(* Logix 5000 project; controller Amvex_Thorpe_Flowmeter vendor 1 type 14 code 106 rev 33.13; software revision 33.01 *)

TASK MainTask (continuous, watchdog 500 ms) : MainProgram
TASK MCP_TESTING_STATION (periodic, rate 10 ms, priority 10, watchdog 500 ms) : MCP_Main
TASK RCP1_FITTING_STATION (periodic, rate 10 ms, priority 10, watchdog 500 ms) : RPC1_Main

MODULES
   Local : vendor 1 type 14 code 106 (Compact 0, rev 33.13)
      RCP1_Valve_Stack : EX260-SEN1 (Ethernet 192.168.30.96, rev 1.1, Output RPI 10 ms)
      MCP_VALVE_STACK : EX260-SEN1 (Ethernet 192.168.30.110, rev 1.1, Output RPI 10 ms)
           MCP_VALVE_STACK:O.OutputArea[0].10   // VB1.O.Sol_A.5
           MCP_VALVE_STACK:O.OutputArea[0].0   // VB1.O.Sol_A.0
           MCP_VALVE_STACK:O.OutputArea[0].1   // VB1.O.Sol_B.0
           MCP_VALVE_STACK:O.OutputArea[0].2   // VB1.O.Sol_A.1
           MCP_VALVE_STACK:O.OutputArea[0].3   // VB1.O.Sol_B.1
           MCP_VALVE_STACK:O.OutputArea[0].4   // VB1.O.Sol_A.2
           MCP_VALVE_STACK:O.OutputArea[0].5   // VB1.O.Sol_B.2
           MCP_VALVE_STACK:O.OutputArea[0].6   // VB1.O.Sol_A.3
           MCP_VALVE_STACK:O.OutputArea[0].7   // VB1.O.Sol_B.3
           MCP_VALVE_STACK:O.OutputArea[0].8   // VB1.O.Sol_A.4
           MCP_VALVE_STACK:O.OutputArea[0].9   // VB1.O.Sol_B.4
           MCP_VALVE_STACK:O.OutputArea[1].0   // VB1.O.Sol_A.8
           MCP_VALVE_STACK:O.OutputArea[1].1   // VB1.O.Sol_B.8
           MCP_VALVE_STACK:O.OutputArea[0].11   // VB1.O.Sol_B.5
           MCP_VALVE_STACK:O.OutputArea[0].12   // VB1.O.Sol_A.6
           MCP_VALVE_STACK:O.OutputArea[0].13   // VB1.O.Sol_B.6
           MCP_VALVE_STACK:O.OutputArea[0].14   // VB1.O.Sol_A.7
           MCP_VALVE_STACK:O.OutputArea[0].15   // VB1.O.Sol_B.7
           MCP_VALVE_STACK:O.OutputArea[1].2   // VB1.O.Sol_A.9
           MCP_VALVE_STACK:O.OutputArea[1].3   // VB1.O.Sol_B.9
      MCP_00 : 1334920000 (Ethernet 192.168.30.101, rev 1.6, StandardDataDriven RPI 10 ms)   // MCP - RR00 - ADAPTER MODULE 00
      Knob_Turner : SV2-CM-ENETIP (Ethernet 192.168.30.115, rev 1.1, StandardDataDriven RPI 10 ms)
           Knob_Turner:I.Data[4]   // Path Status
           Knob_Turner:I.Data[3].4   // Target position reached
           Knob_Turner:I.Data[3].5   // Torque limit active
           Knob_Turner:I.Data[0]   // Torque Feedback
           Knob_Turner:I.Data[1]   // Speed Feedback
           Knob_Turner:I.Data[2]   // Position Error
           Knob_Turner:I.Data[3].2   // Zero Speed
           Knob_Turner:I.Data[3].1   // Servo ON
           Knob_Turner:I.Data[3].0   // Ready
           Knob_Turner:I.Data[3].3   // Target speed reached
           Knob_Turner:I.Data[3].9   // Early overload warnining
           Knob_Turner:I.Data[3]   // General Outputs
           Knob_Turner:I.Data[3].6   // Alarm
           Knob_Turner:I.Data[3].8   // Home Complete
           Knob_Turner:I.Data[3].10   // Warning
           Knob_Turner:I.Data[3].7   // Brake
           Knob_Turner:O.Data[2].1   // Pulse clear
           Knob_Turner:O.Data[3]   // Path target
           Knob_Turner:O.Data[7]   // Path 1 data
           Knob_Turner:O.Data[8]   // Path 2 data
           Knob_Turner:O.Data[2].4   // Alarm reset
           Knob_Turner:O.Data[9]   // Path 3 data
           Knob_Turner:O.Data[2]   // DI control
           Knob_Turner:O.Data[2].7   // Motor Stop
           Knob_Turner:O.Data[2].0   // Servo on
           Knob_Turner:O.Data[2].2   // Torque 1
           Knob_Turner:O.Data[2].3   // Torque 2
           Knob_Turner:O.Data[4]   // Path trigger
           Knob_Turner:O.Data[1]   // DI control switch
           Knob_Turner:O.Data[2].5   // Rev inhibit limit
           Knob_Turner:O.Data[2].6   // Forw inhitibit limit
           Knob_Turner:O.Data[5]   // Speed 1
           Knob_Turner:O.Data[11]   // Torque limit 1
           Knob_Turner:O.Data[12]   // Torque limit 2
           Knob_Turner:O.Data[0]   // Aux functions
           Knob_Turner:O.Data[10]   // Path 4 data
           Knob_Turner:O.Data[6]   // Speed 2
      MCP_SAFETY_CTL : XS26 SC26 SC10 (Ethernet 192.168.30.104, rev 2.1, StandardDataDriven RPI 100 ms, StandardDataDriven RPI 100 ms)
      RCP1_SAFETY_CTL : XS26 SC26 SC10 (Ethernet 192.168.30.93, rev 2.1, StandardDataDriven RPI 100 ms, StandardDataDriven RPI 100 ms)
      IV3 : IV3 Series (Ethernet 192.168.30.106, rev 1.1, StandardDataDriven RPI 25 ms)
           IV3:I.Data[134]   // Tool 10 number of pitches, color average V (brightness), brightness average
           IV3:I.Data[0].1   // Master image regestration response
           IV3:I.Data[144]   // Tool 11 number of pitches, color average V (brightness), brightness average
           IV3:I.Data[154]   // Tool 12 number of pitches, color average V (brightness), brightness average
           IV3:I.Data[36]   // Tool 1 matching rate
           IV3:I.Data[46]   // Tool 2 matching rate
           IV3:I.Data[164]   // Tool 13 number of pitches, color average V (brightness), brightness average
           IV3:I.Data[174]   // Tool 14 number of pitches, color average V (brightness), brightness average
           IV3:I.Data[44]   // Tool 1 number of pitches, color average V (brightness), brightness average
           IV3:I.Data[56]   // Tool 3 matching rate
           IV3:I.Data[42]   // Tool 1 pitch present value MAX, color average H (hue)
           IV3:I.Data[52]   // Tool 2 pitch present value MAX, color average H (hue)
           IV3:I.Data[104]   // Tool 7 number of pitches, color average V (brightness), brightness average
           IV3:I.Data[0].15   // Setting value change failed
           IV3:I.Data[1].12   // Insufficient free space on SD card
           IV3:I.Data[2].0   // Overall judgment OK
           IV3:I.Data[129]   // Tool 10 lower threshold
           IV3:I.Data[130]   // Tool 10 upper threshold
           IV3:I.Data[12]   // Processing time MAX
           IV3:I.Data[0].3   // Warning clear response
           IV3:I.Data[100]   // Tool 7 upper threshold
           IV3:I.Data[26]   // Position adjustment tool matching rate
           IV3:I.Data[20]   // Number of NGs (standard mode/sorting mode)
           IV3:I.Data[21]   // Number of NGs (standard mode/sorting mode)
           IV3:I.Data[15]   // Reserved
           IV3:I.Data[24]   // Reserved
           IV3:I.Data[25]   // Reserved
           IV3:I.Data[30]   // Reserved
           IV3:I.Data[31]   // Reserved
           IV3:I.Data[32]   // Reserved
           IV3:I.Data[66]   // Tool 4 matching rate
           IV3:I.Data[109]   // Tool 8 lower threshold
           IV3:I.Data[110]   // Tool 8 upper threshold
           IV3:I.Data[43]   // Tool 1 pitch present value MIN, color average S (saturation)
           IV3:I.Data[33]   // Reserved
           IV3:I.Data[76]   // Tool 5 matching rate
           IV3:I.Data[119]   // Tool 9 lower threshold
           IV3:I.Data[120]   // Tool 9 upper threshold
           IV3:I.Data[41]   // Tool 1 decimal point position
           IV3:I.Data[53]   // Tool 2 pitch present value MIN, color average S (saturation)
           IV3:I.Data[34]   // Reserved
           IV3:I.Data[86]   // Tool 6 matching rate
           IV3:I.Data[51]   // Tool 2 decimal point position
           IV3:I.Data[63]   // Tool 3 pitch present value MIN, color average S (saturation)
           IV3:I.Data[54]   // Tool 2 number of pitches, color average V (brightness), brightness average
           IV3:I.Data[35]   // Reserved
           IV3:I.Data[96]   // Tool 7 matching rate
           IV3:I.Data[1].1   // Result update complete
           IV3:I.Data[22]   // Number of trigger errors
           IV3:I.Data[2].1   // Position correction
           IV3:I.Data[61]   // Tool 3 decimal point position
           IV3:I.Data[62]   // Tool 3 pitch present value MAX, color average H (hue)
           IV3:I.Data[64]   // Tool 3 number of pitches, color average V (brightness), brightness average
           IV3:I.Data[3].0   // Tool 1
           IV3:I.Data[23]   // Number of trigger errors
           IV3:I.Data[37]   // Tool 1 matching rate MAX
           IV3:I.Data[106]   // Tool 8 matching rate
           IV3:I.Data[116]   // Tool 9 matching rate
           IV3:I.Data[71]   // Tool 4 decimal point position
           IV3:I.Data[73]   // Tool 4 pitch present value MIN, color average S (saturation)
           IV3:I.Data[74]   // Tool 4 number of pitches, color average V (brightness), brightness average
           IV3:I.Data[3].1   // Tool 2
           IV3:I.Data[13]   // Processing time MIN
           IV3:I.Data[38]   // Tool 1 matching rate MIN
           IV3:I.Data[47]   // Tool 2 matching rate MAX
           IV3:I.Data[39]   // Tool 1 lower threshold
           IV3:I.Data[40]   // Tool 1 upper threshold
           IV3:I.Data[81]   // Tool 5 decimal point position
           IV3:I.Data[72]   // Tool 4 pitch present value MAX, color average H (hue)
           IV3:I.Data[3].2   // Tool 3
           IV3:I.Data[48]   // Tool 2 matching rate MIN
           IV3:I.Data[57]   // Tool 3 matching rate MAX
           IV3:I.Data[49]   // Tool 2 lower threshold
           IV3:I.Data[58]   // Tool 3 matching rate MIN
           IV3:I.Data[67]   // Tool 4 matching rate MAX
           IV3:I.Data[68]   // Tool 4 matching rate MIN
           IV3:I.Data[0].7   // Setting value change response
           IV3:I.Data[103]   // Tool 7 pitch present value MIN, color average S (saturation)
           IV3:I.Data[77]   // Tool 5 matching rate MAX
           IV3:I.Data[78]   // Tool 5 matching rate MIN
           IV3:I.Data[0].14   // SD card saving stop failed
           IV3:I.Data[113]   // Tool 8 pitch present value MIN, color average S (saturation)
           IV3:I.Data[0].4   // Statistics reset response
           IV3:I.Data[139]   // Tool 11 lower threshold
           IV3:I.Data[140]   // Tool 11 upper threshold
           IV3:I.Data[101]   // Tool 7 decimal point position
           IV3:I.Data[184]   // Tool 15 number of pitches, color average V (brightness), brightness average
           IV3:I.Data[149]   // Tool 12 lower threshold
           IV3:I.Data[150]   // Tool 12 upper threshold
           IV3:I.Data[111]   // Tool 8 decimal point position
           IV3:I.Data[123]   // Tool 9 pitch present value MIN, color average S (saturation)
           IV3:I.Data[194]   // Tool 16 number of pitches, color average V (brightness), brightness average
           IV3:I.Data[107]   // Tool 8 matching rate MAX
           IV3:I.Data[159]   // Tool 13 lower threshold
           IV3:I.Data[160]   // Tool 13 upper threshold
           IV3:I.Data[121]   // Tool 9 decimal point position
           IV3:I.Data[102]   // Tool 7 pitch present value MAX, color average H (hue)
           IV3:I.Data[133]   // Tool 10 pitch present value MIN, color average S (saturation)
           IV3:I.Data[108]   // Tool 8 matching rate MIN
           IV3:I.Data[127]   // Tool 10 matching rate MAX
           IV3:I.Data[169]   // Tool 14 lower threshold
           IV3:I.Data[170]   // Tool 14 upper threshold
           IV3:I.Data[131]   // Tool 10 decimal point position
           IV3:I.Data[112]   // Tool 8 pitch present value MAX, color average H (hue)
           IV3:I.Data[143]   // Tool 11 pitch present value MIN, color average S (saturation)
           IV3:I.Data[128]   // Tool 10 matching rate MIN
           IV3:I.Data[137]   // Tool 11 matching rate MAX
           IV3:I.Data[179]   // Tool 15 lower threshold
           IV3:I.Data[180]   // Tool 15 upper threshold
           IV3:I.Data[141]   // Tool 11 decimal point position
           IV3:I.Data[122]   // Tool 9 pitch present value MAX, color average H (hue)
           IV3:I.Data[153]   // Tool 12 pitch present value MIN, color average S (saturation)
           IV3:I.Data[138]   // Tool 11 matching rate MIN
           IV3:I.Data[147]   // Tool 12 matching rate MAX
           IV3:I.Data[189]   // Tool 16 lower threshold
           IV3:I.Data[190]   // Tool 16 upper threshold
           IV3:I.Data[151]   // Tool 12 decimal point position
           IV3:I.Data[132]   // Tool 10 pitch present value MAX, color average H (hue)
           IV3:I.Data[163]   // Tool 13 pitch present value MIN, color average S (saturation)
           IV3:I.Data[148]   // Tool 12 matching rate MIN
           IV3:I.Data[157]   // Tool 13 matching rate MAX
           IV3:I.Data[1].13   // Buffer overrun status
           IV3:I.Data[6]   // Number of remaining buffers
           IV3:I.Data[161]   // Tool 13 decimal point position
           IV3:I.Data[142]   // Tool 11 pitch present value MAX, color average H (hue)
           IV3:I.Data[173]   // Tool 14 pitch present value MIN, color average S (saturation)
           IV3:I.Data[196]   // master number/total status product type
           IV3:I.Data[0].5   // Buffer clear response
           IV3:I.Data[158]   // Tool 13 matching rate MIN
           IV3:I.Data[167]   // Tool 14 matching rate MAX
           IV3:I.Data[87]   // Tool 6 matching rate MAX
           IV3:I.Data[88]   // Tool 6 matching rate MIN
           IV3:I.Data[171]   // Tool 14 decimal point position
           IV3:I.Data[152]   // Tool 12 pitch present value MAX, color average H (hue)
           IV3:I.Data[183]   // Tool 15 pitch present value MIN, color average S (saturation)
           IV3:I.Data[126]   // Tool 10 matching rate
           IV3:I.Data[168]   // Tool 14 matching rate MIN
           IV3:I.Data[177]   // Tool 15 matching rate MAX
           IV3:I.Data[97]   // Tool 7 matching rate MAX
           IV3:I.Data[9]   // Program No. during judgment
           IV3:I.Data[181]   // Tool 15 decimal point position
           IV3:I.Data[162]   // Tool 13 pitch present value MAX, color average H (hue)
           IV3:I.Data[193]   // Tool 16 pitch present value MIN, color average S (saturation)
           IV3:I.Data[114]   // Tool 8 number of pitches, color average V (brightness), brightness average
           IV3:I.Data[136]   // Tool 11 matching rate
           IV3:I.Data[178]   // Tool 15 matching rate MIN
           IV3:I.Data[187]   // Tool 16 matching rate MAX
           IV3:I.Data[98]   // Tool 7 matching rate MIN
           IV3:I.Data[191]   // Tool 16 decimal point position
           IV3:I.Data[172]   // Tool 14 pitch present value MAX, color average H (hue)
           IV3:I.Data[83]   // Tool 5 pitch present value MIN, color average S (saturation)
           IV3:I.Data[146]   // Tool 12 matching rate
           IV3:I.Data[188]   // Tool 16 matching rate MIN
           IV3:I.Data[117]   // Tool 9 matching rate MAX
           IV3:I.Data[156]   // Tool 13 matching rate
           IV3:I.Data[166]   // Tool 14 matching rate
           IV3:I.Data[1].7   // SD card identification status
           IV3:I.Data[182]   // Tool 15 pitch present value MAX, color average H (hue)
           IV3:I.Data[82]   // Tool 5 pitch present value MAX, color average H (hue)
           IV3:I.Data[176]   // Tool 15 matching rate
           IV3:I.Data[186]   // Tool 16 matching rate
           IV3:I.Data[18]   // OK count (standard mode) Total sort count (sorting mode)
           IV3:I.Data[93]   // Tool 6 pitch present value MIN, color average S (saturation)
           IV3:I.Data[118]   // Tool 9 matching rate MIN
           IV3:I.Data[50]   // Tool 2 upper threshold
           IV3:I.Data[91]   // Tool 6 decimal point position
           IV3:I.Data[0].6   // SD card saving stop response
           IV3:I.Data[27]   // Position adjustment tool matching rate MAX
           IV3:I.Data[0].11   // Reserved
           IV3:I.Data[0].12   // Reserved
           IV3:I.Data[0].0   // Trigger response
           IV3:I.Data[16]   // Number of triggers
           IV3:I.Data[17]   // Number of triggers
           IV3:I.Data[1].0   // Result available
           IV3:I.Data[59]   // Tool 3 lower threshold
           IV3:I.Data[60]   // Tool 3 upper threshold
           IV3:I.Data[69]   // Tool 4 lower threshold
           IV3:I.Data[70]   // Tool 4 upper threshold
           IV3:I.Data[79]   // Tool 5 lower threshold
           IV3:I.Data[80]   // Tool 5 upper threshold
           IV3:I.Data[89]   // Tool 6 lower threshold
           IV3:I.Data[2].6   // Overall judgment NG
           IV3:I.Data[1].14   // Warning status
           IV3:I.Data[0].8   // Trigger failed
           IV3:I.Data[0].9   // Master image regestration failed
           IV3:I.Data[29]   // Position adjustment tool threshold
           IV3:I.Data[3].3   // Tool 4
           IV3:I.Data[1].15   // Error status
           IV3:I.Data[3].4   // Tool 5
           IV3:I.Data[3].5   // Tool 6
           IV3:I.Data[3].6   // Tool 7
           IV3:I.Data[3].7   // Tool 8
           IV3:I.Data[14]   // Processing time AVE
           IV3:I.Data[8]   // Current Program No.
           IV3:I.Data[3].8   // Tool 9
           IV3:I.Data[45]   // Reserved
           IV3:I.Data[4]   // Error code
           IV3:I.Data[55]   // Reserved
           IV3:I.Data[65]   // Reserved
           IV3:I.Data[75]   // Reserved
           IV3:I.Data[85]   // Reserved
           IV3:I.Data[1].3   // Imaging
           IV3:I.Data[2].2   // Logic 1
           IV3:I.Data[2].3   // Logic 2
           IV3:I.Data[0].13   // Reserved
           IV3:I.Data[1].10   // Reserved
           IV3:I.Data[1].11   // Reserved
           IV3:I.Data[2].4   // Logic 3
           IV3:I.Data[0].10   // Program switching failed
           IV3:I.Data[0].2   // Program switching response
           IV3:I.Data[105]   // Reserved
           IV3:I.Data[2].10   // Reserved
           IV3:I.Data[95]   // Reserved
           IV3:I.Data[2].11   // Reserved
           IV3:I.Data[2].5   // Logic 4
           IV3:I.Data[3].9   // Tool 10
           IV3:I.Data[2].12   // Reserved
           IV3:I.Data[2].13   // Reserved
           IV3:I.Data[2].14   // Reserved
           IV3:I.Data[3].10   // Tool 11
           IV3:I.Data[2].15   // Reserved
           IV3:I.Data[1].4   // RUN
           IV3:I.Data[10]   // Result No.
           IV3:I.Data[115]   // Reserved
           IV3:I.Data[125]   // Reserved
           IV3:I.Data[135]   // Reserved
           IV3:I.Data[145]   // Reserved
           IV3:I.Data[155]   // Reserved
           IV3:I.Data[165]   // Reserved
           IV3:I.Data[175]   // Reserved
           IV3:I.Data[185]   // Reserved
           IV3:I.Data[195]   // Reserved
           IV3:I.Data[1].2   // Busy
           IV3:I.Data[7]   // Checksum
           IV3:I.Data[192]   // Tool 16 pitch present value MAX, color average H (hue)
           IV3:I.Data[28]   // Position adjustment tool matching rate MIN
           IV3:I.Data[19]   // OK count (standard mode) Total sort count (sorting mode)
           IV3:I.Data[92]   // Tool 6 pitch present value MAX, color average H (hue)
           IV3:I.Data[3].11   // Tool 12
           IV3:I.Data[1].6   // Reserved
           IV3:I.Data[11]   // Processing time
           IV3:I.Data[1].9   // Reserved
           IV3:I.Data[84]   // Tool 5 number of pitches, color average V (brightness), brightness average
           IV3:I.Data[3].12   // Tool 13
           IV3:I.Data[94]   // Tool 6 number of pitches, color average V (brightness), brightness average
           IV3:I.Data[1].5   // Ready
           IV3:I.Data[3].13   // Tool 14
           IV3:I.Data[2].7   // Reserved
           IV3:I.Data[2].8   // Reserved
           IV3:I.Data[2].9   // Reserved
           IV3:I.Data[5]   // Warning code
           IV3:I.Data[3].14   // Tool 15
           IV3:I.Data[124]   // Tool 9 number of pitches, color average V (brightness), brightness average
           IV3:I.Data[3].15   // Tool 16
           IV3:I.Data[90]   // Tool 6 upper threshold
           IV3:I.Data[99]   // Tool 7 lower threshold
           IV3:I.Data[1].8   // Sorting mode information
           IV3:O.Data[0].10   // Reserved
           IV3:O.Data[0].11   // Reserved
           IV3:O.Data[0].12   // Reserved
           IV3:O.Data[0].13   // Reserved
           IV3:O.Data[0].14   // Reserved
           IV3:O.Data[1].0   // Result acquisition complete notification
           IV3:O.Data[0].6   // SD card saving stop request
           IV3:O.Data[0].5   // Buffer clear request
           IV3:O.Data[0].7   // Setting value change request
           IV3:O.Data[0].2   // Program switching request
           IV3:O.Data[4]   // Upper/lower limit/Master Text/FTP/SD saving settings
           IV3:O.Data[0].4   // Statistics reset request
           IV3:O.Data[5]   // Upper/lower limit/Master Text/FTP/SD saving settings
           IV3:O.Data[0].3   // Warning clear request
           IV3:O.Data[0].15   // Reserved
           IV3:O.Data[3]   // Upper/lower limit setting No./Master text setting No./FTP/Sdsaved setting No.
           IV3:O.Data[0].1   // Master image registration request
           IV3:O.Data[1].10   // Reserved
           IV3:O.Data[1].11   // Reserved
           IV3:O.Data[1].12   // Reserved
           IV3:O.Data[1].13   // Reserved
           IV3:O.Data[1].14   // Reserved
           IV3:O.Data[1].15   // Reserved
           IV3:O.Data[2]   // Program number
           IV3:O.Data[0].0   // Trigger request
           IV3:O.Data[0].8   // Reserved
           IV3:O.Data[0].9   // Reserved
           IV3:O.Data[1].1   // Reserved
           IV3:O.Data[1].2   // Reserved
           IV3:O.Data[1].3   // Reserved
           IV3:O.Data[1].4   // Reserved
           IV3:O.Data[1].5   // Reserved
           IV3:O.Data[1].6   // Reserved
           IV3:O.Data[1].7   // Reserved
           IV3:O.Data[1].8   // Reserved
           IV3:O.Data[1].9   // Reserved
      SR : SR-2000 (Ethernet 192.168.30.108, rev 1.1, StandardDataDriven RPI 20 ms)
           SR:I.Data[0].2   // Result Data Strobe
           SR:I.Data[20]   // Register Preset Data Result Code
           SR:I.Data[21]   // Register Preset Data Result Code
           SR:I.Data[2].2   // Register Preset Data Complete
           SR:I.Data[10]   // ISO/IEC15415 Grade
           SR:I.Data[38]   // Result Data Update Count
           SR:I.Data[2].7   // External Request Complete
           SR:I.Data[16]   // Read Result Code
           SR:I.Data[30]   // External Request Result Code
           SR:I.Data[3].2   // Register Preset Data Failure
           SR:I.Data[40]   // Trigger Input Count for Master
           SR:I.Data[14]   // ISO/IEC15416 Grade
           SR:I.Data[39]   // Result Data Update Count
           SR:I.Data[41]   // Trigger Input Count for Master
           SR:I.Data[1].4   // Error Busy
           SR:I.Data[5].1   // Matching Level Unstable
           SR:I.Data[18]   // Preset Result Code
           SR:I.Data[17]   // Read Result Code
           SR:I.Data[5].4   // ADE AS9132 Unstable
           SR:I.Data[8]   // Matching Level
           SR:I.Data[11]   // Reserved
           SR:I.Data[13]   // Reserved
           SR:I.Data[15]   // Reserved
           SR:I.Data[26]   // Reserved
           SR:I.Data[27]   // Reserved
           SR:I.Data[28]   // Reserved
           SR:I.Data[29]   // Reserved
           SR:I.Data[34]   // Slave ID
           SR:I.Data[19]   // Preset Result Code
           SR:I.Data[32]   // General Error Code
           SR:I.Data[35]   // Slave ID
           SR:I.Data[0].1   // Result Data Available
           SR:I.Data[0].6   // Buffer Overflow Error
           SR:I.Data[36]   // Result Data Ready Count
           SR:I.Data[37]   // Result Data Ready Count
           SR:I.Data[3].7   // External Request Failure
           SR:I.Data[5].2   // ISO/IEC15415 Unstable
           SR:I.Data[5].5   // ISO/IEC15416 Unstable
           SR:I.Data[1].0   // Busy
           SR:I.Data[0].3   // Reserved
           SR:I.Data[33]   // General Error Code
           SR:I.Data[0].4   // Reserved
           SR:I.Data[5].3   // AIM DPM Unstable
           SR:I.Data[0].5   // Reserved
           SR:I.Data[1].5   // Reserved
           SR:I.Data[1].7   // Reserved
           SR:I.Data[2].5   // Reserved
           SR:I.Data[2].6   // Reserved
           SR:I.Data[3].5   // Reserved
           SR:I.Data[3].6   // Reserved
           SR:I.Data[4].2   // Reserved
           SR:I.Data[4].3   // Reserved
           SR:I.Data[4].7   // Reserved
           SR:I.Data[5].0   // Unstable
           SR:I.Data[1].2   // Lock Busy
           SR:I.Data[22]   // Tune Result Code
           SR:I.Data[23]   // Tune Result Code
           SR:I.Data[2].4   // Bload Complete
           SR:I.Data[3].1   // Preset Failure
           SR:I.Data[42]   // Result Data Size
           SR:I.Data[43]   // Result Data Size
           SR:I.Data[4].0   // Input 1 Status
           SR:I.Data[4].1   // Input 2 Status
           SR:I.Data[24]   // Bload Result Code
           SR:I.Data[25]   // Bload Result Code
           SR:I.Data[2].1   // Preset Complete
           SR:I.Data[4].4   // Output 1 Status
           SR:I.Data[4].5   // Output 2 Status
           SR:I.Data[4].6   // Output 3 Status
           SR:I.Data[6]   // Reserved
           SR:I.Data[1].3   // Mode Busy
           SR:I.Data[5].6   // Reserved
           SR:I.Data[5].7   // Reserved
           SR:I.Data[44]   // Result Data
           SR:I.Data[45]   // Result Data
           SR:I.Data[7]   // Reserved
           SR:I.Data[31]   // External Request Result Code
           SR:I.Data[46]   // Result Data
           SR:I.Data[47]   // Result Data
           SR:I.Data[48]   // Result Data
           SR:I.Data[49]   // Result Data
           SR:I.Data[50]   // Result Data
           SR:I.Data[0].7   // General Error
           SR:I.Data[2].0   // Read Complete
           SR:I.Data[2].3   // Tune Complete
           SR:I.Data[0].0   // Error
           SR:I.Data[12]   // AIM DPM Grade
           SR:I.Data[1].1   // Trigger Busy
           SR:I.Data[9]   // Reserved
           SR:I.Data[3].4   // Bload Failure
           SR:I.Data[1].6   // Ready
           SR:I.Data[3].0   // Read Failure
           SR:I.Data[3].3   // Tune Failure
           SR:O.Data[2].2   // Register Preset Data Complete Clear
           SR:O.Data[12]   // User Data
           SR:O.Data[1].1   // Preset Request
           SR:O.Data[2].0   // Read Complete Clear
           SR:O.Data[2].1   // Preset Complete Clear
           SR:O.Data[1].2   // Register Preset Data Request
           SR:O.Data[13]   // User Data
           SR:O.Data[3]   // Reserved
           SR:O.Data[2].3   // Tune Complete Clear
           SR:O.Data[14]   // User Data
           SR:O.Data[15]   // User Data
           SR:O.Data[16]   // User Data
           SR:O.Data[17]   // User Data
           SR:O.Data[6]   // Reserved
           SR:O.Data[4]   // Bank Number
           SR:O.Data[7]   // Reserved
           SR:O.Data[8]   // Reserved
           SR:O.Data[0].0   // Reserved
           SR:O.Data[0].1   // Result Data Latch
           SR:O.Data[2].7   // External Request Complete Clear
           SR:O.Data[2].4   // Bload Complete Clear
           SR:O.Data[0].2   // Reserved
           SR:O.Data[0].3   // Reserved
           SR:O.Data[0].4   // Reserved
           SR:O.Data[0].5   // Reserved
           SR:O.Data[0].6   // Reserved
           SR:O.Data[1].5   // Reserved
           SR:O.Data[1].6   // Reserved
           SR:O.Data[9]   // Reserved
           SR:O.Data[1].7   // Reserved
           SR:O.Data[2].5   // Reserved
           SR:O.Data[2].6   // Reserved
           SR:O.Data[5]   // Bank Number
           SR:O.Data[10]   // User Data Size
           SR:O.Data[1].4   // Bload Request
           SR:O.Data[0].7   // Error Clear
           SR:O.Data[11]   // User Data Size
           SR:O.Data[1].0   // Read Request
           SR:O.Data[1].3   // Tune Request
      Conv : OPC-2-ETHIG-IN (Ethernet 192.168.30.107, rev 2.1, StandardDataDriven RPI 100 ms)
           Conv:I.Data[0].6   // READY
           Conv:O.Data[0].0   // RUN
      LPM100 : 0496_000C_0002 (Ethernet 192.168.30.103, rev 1.2, StandardDataDriven RPI 20 ms)
      RCP1_00 : 1334920000 (Ethernet 192.168.30.87, rev 1.6, StandardDataDriven RPI 10 ms)
           RCP1_00:I1.ConnectionFaulted   // IO rack comms
      LPM5 : 0496_000C_0002 (Ethernet 192.168.30.102, rev 1.2, StandardDataDriven RPI 20 ms)
END_MODULES

TYPE Alicat :
STRUCT
   Enable : BOOL;
   Test : BOOL;
   CMD_AOI : AlicatCommand;
   Input_AOI : AlicatUpdateInput;
   IoData : AlicatIoData;
   CmdData : INT[2];
   Oxygen : Oxygen;
   Ready : BOOL;
   Flow : REAL;
   Flow_Avg : REAL;
   Flow_data : REAL[25];
   Flow_TM1 : TIMER;
   Flow_TM2 : TIMER;
   Flow_Data_Inc : INT;
   Upper_Lim_Num : REAL;
   Lower_Lim_Num : REAL;
END_STRUCT
END_TYPE

TYPE AlicatIoData :
STRUCT
   Status : DINT;   // Device Status Flags
   T_OVER : BOOL;   // Temperature Overflow
   T_UNDR : BOOL;   // Temperature Underflow
   V_OVER : BOOL;   // Volumetric Overflow
   V_UNDR : BOOL;   // Volumetric Underflow
   M_OVER : BOOL;   // Mass Overflow
   M_UNDR : BOOL;   // Mass Underflow
   P_OVER : BOOL;   // Pressure Overflow
   TOT_OVER : BOOL;   // Totalizer Overflow
   HLD : BOOL;   // PID Loop in Hold
   ADC : BOOL;   // ADC Error
   EXH : BOOL;   // PID Exhaust
   OPL : BOOL;   // Over Pressure Limit
   TMF : BOOL;   // Flow Overflow During Totalize
   Pressure : REAL;
   Temperature : REAL;
   VolFlow : REAL;
   MassFlow : REAL;
   ActualSetpoint : REAL;
   ValveDrivePct : REAL;
   Totalizer : REAL;
   RequestedSetpoint : REAL;
   GasIndex : INT;
   Config : SINT;
   PRESS : BOOL;   // Pressure Reading Valid
   TEMP : BOOL;   // Temperature Reading Valid
   VFLOW : BOOL;   // Volumetric Flow Reading Valid
   MFLOW : BOOL;   // Mass Flow Reading Valid
   SP : BOOL;   // Setpoint Reading Valid
   VDRIVE : BOOL;   // Valve Drive Percentage Reading Valid
   TOTAL : BOOL;   // Totalizer Reading Valid
END_STRUCT
END_TYPE

TYPE Auto_seq :
STRUCT
   Next_Step : DINT;
   Current_Step : DINT;
END_STRUCT
END_TYPE

TYPE Banner_Fault_Log_UDT :
STRUCT
   Time_Stamp : DINT;
   Name_Length : DINT;
   Name : SINT[12];
   Error_Code : INT;
   Advanced_Error_Code : INT;
   Error_Index : INT;
   Reserved : DINT;
END_STRUCT
END_TYPE

TYPE Barcode :
STRUCT
   Ready : BOOL;
   Result : STRING;
   Read : BOOL;
   Result_avalible : BOOL;
   Read_complete : BOOL;
   Read_complete_clear : BOOL;
   Read_success : BOOL;
   Read_failed : BOOL;
END_STRUCT
END_TYPE

TYPE Conv :
STRUCT
   VFD : VFD;
   Stop : Stop[5];
   Lift : Lift;
   Diverter : Diverter;
   Drop_TM : TIMER[3];
   Downstream_Full : AOI_DIG_INPUT_DEB;
   Reject_Full : AOI_DIG_INPUT_DEB;
END_STRUCT
END_TYPE

TYPE Diverter :
STRUCT
   Ext : BOOL;
   Ret : BOOL;
   Present : AOI_DIG_INPUT_DEB;
END_STRUCT
END_TYPE

TYPE Driver :
STRUCT
   Ext : BOOL;
   Ret : BOOL;
   Extd : AOI_DIG_INPUT_DEB;
   Retd : AOI_DIG_INPUT_DEB;
   Drive_TM : TIMER;
END_STRUCT
END_TYPE

TYPE FastTest :
STRUCT
   Ext : BOOL;
   Ret : BOOL;
   Extd : AOI_DIG_INPUT_DEB;
   Retd : AOI_DIG_INPUT_DEB;
   Outlet_Seal : BOOL;
   Outlet_Unseal : BOOL;
   Inlet_Seal : BOOL;
   Inlet_Unseal : BOOL;
END_STRUCT
END_TYPE

TYPE HMI :
STRUCT
   Conv : Conv;
   Testing : Testing;
   Part_Count : DINT;
   Lifetime_Part_Count : REAL;
   Fault_AOI : FAULT_AOI[32];
   Fault : DINT[2];
   FAULTED : DINT[2];
   HMI : HMI_Temp;
   Performance : REAL;
   UptimeSTM : TIMER;
   UptimeM : COUNTER;
   DowntimeSTM : TIMER;
   DowntimeM : COUNTER;
   Cycle_Time : DINT;
   UptimeH : COUNTER;
   DowntimeH : COUNTER;
   UptimeTM : TIMER;
   Batch_Count : DINT;
   Testing_Status : INT[6];
END_STRUCT
END_TYPE

TYPE HMI_Temp :
STRUCT
   Reset_Counter : BOOL;
   Reset_Faults : BOOL;
   Batch_Number : STRING;
   Needle_Bypass : BOOL;
   Max_Cycle_Time : REAL;
END_STRUCT
END_TYPE

TYPE Homing :
STRUCT
   Testing : Testing;
   Conv : Conv;
END_STRUCT
END_TYPE

TYPE Hood :
STRUCT
   Extd : AOI_DIG_INPUT_DEB;
   Retd : AOI_DIG_INPUT_DEB;
   Ext : BOOL;
   Ret : BOOL;
END_STRUCT
END_TYPE

TYPE Jog :
STRUCT
   Enabled : BOOL;
   X : BOOL[32];
   Y : BOOL[32];
   Z : BOOL[32];
   Stop : BOOL;
   Jog_AOI : MoveLinRelWRF;
   X_Inc : REAL;
   Y_Inc : REAL;
   Z_Inc : REAL;
   Increment : REAL;
   Speed : REAL;
END_STRUCT
END_TYPE

TYPE Knob_Turner :
STRUCT
   Enable : BOOL;
   Ready : BOOL;
   Home : BOOL;
   Speed_Reached : BOOL;
   Alarm : BOOL;
   Path_Status : BOOL;
   Reset : BOOL;
   Stop : BOOL;
   Turn_Open : BOOL;
   Turn_Close : BOOL;
   Turn_2 : BOOL;
   Turn_8 : BOOL;
   Turn_15 : BOOL;
   Turn_Speed : REAL;
   Rapid_Speed : REAL;
   T2_Rapid_Pos : REAL;
   T8_Rapid_Pos : REAL;
   T15_Rapid_Pos : REAL;
   Torque_EN1 : BOOL;
   Torque_EN2 : BOOL;
   Torque1 : REAL;
   Torque2 : REAL;
   Torque_Feedback : REAL;
   Path : REAL;
   Trigger_Path : BOOL;
   Ext : BOOL;
   Ret : BOOL;
   Extd : AOI_DIG_INPUT_DEB;
   Retd : AOI_DIG_INPUT_DEB;
   Grip : BOOL;
   Ungrip : BOOL;
END_STRUCT
END_TYPE

TYPE Lift :
STRUCT
   Stop : Stop;
   Ext : BOOL;
   Ret : BOOL;
   Extd : AOI_DIG_INPUT_DEB;
   Retd : AOI_DIG_INPUT_DEB;
END_STRUCT
END_TYPE

TYPE MCP :
STRUCT
   Conv : Conv;
   Testing : Testing;
   Part_Count : DINT;
   Lifetime_Part_Count : REAL;
   Fault_AOI : FAULT_AOI[100];
   Fault : DINT[2];
   FAULTED : DINT[2];
   HMI_Temp : HMI_Temp;
   Performance : REAL;
   Availability : REAL;
   UptimeSTM : TIMER;
   UptimeM : COUNTER;
   DowntimeSTM : TIMER;
   DowntimeM : COUNTER;
   Cycle_Time : DINT;
   UptimeH : COUNTER;
   DowntimeH : COUNTER;
   UptimeTM : TIMER;
   DowntimeTM : TIMER;
   UptimeS : COUNTER;
   DowntimeS : COUNTER;
   Planned_Production_Time : DINT;
   PPTS : DINT;
   PPTM : DINT;
   PPTH : DINT;
   Batch_Count : DINT;
   HMI : HMI;
   Homing : Homing;
END_STRUCT
END_TYPE

TYPE MODE :
STRUCT
   Auto : BOOL;   // Auto Mode
   Manual : BOOL;   // Manual Mode
   Off : BOOL;   // Off Mode
   Cycle_Start_PB : BOOL;   // Cycle Start Push Button
   Cycle_Stop_PB : BOOL;   // Cycle Stop Push Button
   Auto_PB : BOOL;   // Auto Mode Push Button
   Manual_PB : BOOL;   // Manual Mode Push Button
   AOI : AOI_DIG_INPUT_DEB;
   Manual_ONS : BOOL;   // Manual Mode Oneshot
   Faulted : BOOL;   // Fault Active
   Ready : BOOL;   // Ready to go in to auto
   Homed : BOOL;   // Machine is at Home Position
   Home : BOOL;   // Home the Machine
   Homing : BOOL;   // Machine is Homing
   Selector : INT;   // Control mode via HMI
END_STRUCT
END_TYPE

TYPE Oxygen :
STRUCT
   Oxygen : BOOL;
   To_100LPM : BOOL;
   To_5LPM : BOOL;
END_STRUCT
END_TYPE

TYPE Oxygen_Sys :
STRUCT
   On : BOOL;
   Off : BOOL;
END_STRUCT
END_TYPE

TYPE Part :
STRUCT
   Code : STRING;
   Results : INT;
END_STRUCT
END_TYPE

TYPE RCP1 :
STRUCT
   Inlet_Driver : Driver;
   Needle_Driver : Driver;
   Saftey : Safety;
   Part_Present : AOI_DIG_INPUT_DEB;
   Part_Count : DINT;
   Lifetime_Part_Count : REAL;
   Home_PB : AOI_DIG_INPUT_DEB;
   Select_Switch : AOI_DIG_INPUT_DEB;
   Reset_PB : AOI_DIG_INPUT_DEB;
   Stacklight : Stacklight;
   Fault_AOI : FAULT_AOI[12];
   Fault : DINT;
   FAULTED : DINT;
   Air_Pressure : AOI_DIG_INPUT_DEB;
   HMI : HMI_Temp;
   Max_Cycle_Time : DINT;
   Performance : REAL;
   Availability : REAL;
   UptimeTM : TIMER;
   UptimeS : COUNTER;
   UptimeM : COUNTER;
   UptimeH : COUNTER;
   DowntimeTM : TIMER;
   DowntimeS : COUNTER;
   DowntimeM : COUNTER;
   DowntimeH : COUNTER;
   Planned_Production_Time : DINT;
   PPTS : DINT;
   PPTM : DINT;
   PPTH : DINT;
   Batch_Number : STRING;
   Batch_Count : DINT;
   Needle_Bypass : BOOL;
END_STRUCT
END_TYPE

TYPE Robot :
STRUCT
   Connection : Connect;
   Setup : INT;
   Activate : BOOL;
   Home : BOOL;
   Safe_Home : BOOL;
   Power_Reset : BOOL;
   Reset : BOOL;
   Lin_Speed : REAL;
   Move_to_Knob : BOOL;
   Turn : BOOL;
   Unturn : BOOL;
   Turn_TM : TIMER;
   Turn_Deg : REAL;
   Turn_Speed : REAL;
   Turn_ONS : BOOL;
   MoveLin : BOOL;
   MoveLin_Pos : REAL[6];
   Tool_Position_1 : REAL[6];
   Tool_Position_2 : REAL[6];
   To_Pos_1 : BOOL;
   To_Pos_2 : BOOL;
   At_Pos_1 : BOOL;
   At_Pos_2 : BOOL;
   Pos_1_Set : BOOL;
   Pos_2_Set : BOOL;
   DN : BOOL;
   Reset_Error : BOOL;
   Pause : BOOL;
   Deactivate : BOOL;
   Knob_Torque : REAL;
   Jog : Jog;
   Turn_Speed_AOI : SetJointVel;
   Turn_AOI : MoveJoints;
   ErrorAOI : RobotErrors;
   Torque_Config_AOI : SetTorqueLimitsCfg;
   Torque_Limit_AOI : SetTorqueLimits;
   MoveLin_AOI : MoveLin;
   LinVel_AOI : SetCartLinVel;
   Close : BOOL;
   Open : BOOL;
END_STRUCT
END_TYPE

TYPE Safety :
STRUCT
   Lockout : BOOL;
   Input_Fault : BOOL;
   Output_Fault : BOOL;
   Estop : BOOL;
   Light_Curtain : BOOL;
   Door : BOOL;
   Output : BOOL;
   Reset : BOOL;
   RDC_Active : BOOL;
   RDC_Code : INT;
   RDC_Error : BOOL;
   AOI : Banner_XS26_RCD_Function;
END_STRUCT
END_TYPE

TYPE SEQ :
STRUCT
   Current_Step : INT;   // Current Sequence Step
   Next_Step : INT;   // Next Sequence Step
   Active : BOOL;   // Sequence Active
   Run_Perm : BOOL;   // Sequence Run Permissive
   Cycle_Start : BOOL;   // Cycle Start
   Cycle_Stop : BOOL;   // Cycle Stop
   Cycle_Stopping : BOOL;   // Cycle Stopping
   In_Cycle : BOOL;   // In Cycle
   Single_Step : BOOL;   // Single Step
   Single_Step_Ons : BOOL;   // Single Step Oneshot
   MCP_Reset_PB : BOOL;   // Main Control Panel Reset Pushbutton
   OC_Reset_PB : BOOL;   // Operator Console Reset Pushbutton
   Time_Out : TIMER;   // Sequence Time Out
   Time_Out_Sec : INT;   // Time Out Seconds
   HMI : MODE;
   Reset : BOOL;   // Reset
   HMI_Reset : BOOL;   // HMI Pushbutton
END_STRUCT
END_TYPE

TYPE Stacklight :
STRUCT
   Green : BOOL;
   Yellow : BOOL;
   Red : BOOL;
   Blue : BOOL;
   White : BOOL;
END_STRUCT
END_TYPE

TYPE Stop :
STRUCT
   Present : AOI_DIG_INPUT_DEB;
   Release : BOOL;
   Hold : BOOL;
END_STRUCT
END_TYPE

TYPE Test :
STRUCT
   Flow : REAL;
   Range : REAL;
   Test_TM : TIMER;
   Time : INT;
END_STRUCT
END_TYPE

TYPE Testing :
STRUCT
   Robot : Robot;
   FastTest : FastTest;
   Hood : Hood;
   Alicat : Alicat[2];
   Vision : Vision;
   Barcode : Barcode;
   Part_Present : AOI_DIG_INPUT_DEB;
   Saftey : Safety;
   Air_pressure : AOI_DIG_INPUT_DEB;
   Stacklight : Stacklight;
   Part : Part[100];
   Test : Test[7];
   Load_PB : AOI_DIG_INPUT_DEB;
   Oxygen_Sys : Oxygen_Sys;
   Knob_Turner : Knob_Turner;
   Reject_Pallet : BOOL;
END_STRUCT
END_TYPE

TYPE UDT_015_Data_I :   // UR20_FBC_EIP Module UR20_FBC_EIP UDT for UR20_16DI_P Order No.: 1315200000 Process Data (Inputs)
STRUCT
   Ch_00 : BOOL;   // UR20_16DI_P Process Data Ch_00
   Ch_01 : BOOL;   // UR20_16DI_P Process Data Ch_01
   Ch_02 : BOOL;   // UR20_16DI_P Process Data Ch_02
   Ch_03 : BOOL;   // UR20_16DI_P Process Data Ch_03
   Ch_04 : BOOL;   // UR20_16DI_P Process Data Ch_04
   Ch_05 : BOOL;   // UR20_16DI_P Process Data Ch_05
   Ch_06 : BOOL;   // UR20_16DI_P Process Data Ch_06
   Ch_07 : BOOL;   // UR20_16DI_P Process Data Ch_07
   Ch_08 : BOOL;   // UR20_16DI_P Process Data Ch_08
   Ch_09 : BOOL;   // UR20_16DI_P Process Data Ch_09
   Ch_10 : BOOL;   // UR20_16DI_P Process Data Ch_10
   Ch_11 : BOOL;   // UR20_16DI_P Process Data Ch_11
   Ch_12 : BOOL;   // UR20_16DI_P Process Data Ch_12
   Ch_13 : BOOL;   // UR20_16DI_P Process Data Ch_13
   Ch_14 : BOOL;   // UR20_16DI_P Process Data Ch_14
   Ch_15 : BOOL;   // UR20_16DI_P Process Data Ch_15
END_STRUCT
END_TYPE

TYPE UDT_015_I :   // UR20_FBC_EIP Module UR20_FBC_EIP UDT for UR20_16DI_P Order No.: 1315200000 generic Module Data (Inputs)
STRUCT
   Data : UDT_015_Data_I;   // UR20_16DI_P generic Module Data Data
   Diagnostic : UDT_Diagnostic;   // UR20_16DI_P generic Module Data Diagnostic
   ProcessAlarm : UDT_ProcessAlarm;   // UR20_16DI_P generic Module Data ProcessAlarm
   StatusDiagAlarm : BOOL;   // UR20_16DI_P generic Module Data StatusDiagAlarm
   StatusProcessAlarm : BOOL;   // UR20_16DI_P generic Module Data StatusProcessAlarm
END_STRUCT
END_TYPE

TYPE UDT_020_Data_O :   // UR20_FBC_EIP Module UR20_FBC_EIP UDT for UR20_16DO_P Order No.: 1315250000 Process Data (Outputs)
STRUCT
   Ch_00 : BOOL;   // UR20_16DO_P Process Data Ch_00
   Ch_01 : BOOL;   // UR20_16DO_P Process Data Ch_01
   Ch_02 : BOOL;   // UR20_16DO_P Process Data Ch_02
   Ch_03 : BOOL;   // UR20_16DO_P Process Data Ch_03
   Ch_04 : BOOL;   // UR20_16DO_P Process Data Ch_04
   Ch_05 : BOOL;   // UR20_16DO_P Process Data Ch_05
   Ch_06 : BOOL;   // UR20_16DO_P Process Data Ch_06
   Ch_07 : BOOL;   // UR20_16DO_P Process Data Ch_07
   Ch_08 : BOOL;   // UR20_16DO_P Process Data Ch_08
   Ch_09 : BOOL;   // UR20_16DO_P Process Data Ch_09
   Ch_10 : BOOL;   // UR20_16DO_P Process Data Ch_10
   Ch_11 : BOOL;   // UR20_16DO_P Process Data Ch_11
   Ch_12 : BOOL;   // UR20_16DO_P Process Data Ch_12
   Ch_13 : BOOL;   // UR20_16DO_P Process Data Ch_13
   Ch_14 : BOOL;   // UR20_16DO_P Process Data Ch_14
   Ch_15 : BOOL;   // UR20_16DO_P Process Data Ch_15
END_STRUCT
END_TYPE

TYPE UDT_020_I :   // UR20_FBC_EIP Module UR20_FBC_EIP UDT for UR20_16DO_P Order No.: 1315250000 generic Module Data (Inputs)
STRUCT
   Diagnostic : UDT_Diagnostic;   // UR20_16DO_P generic Module Data Diagnostic
   ProcessAlarm : UDT_ProcessAlarm;   // UR20_16DO_P generic Module Data ProcessAlarm
   StatusDiagAlarm : BOOL;   // UR20_16DO_P generic Module Data StatusDiagAlarm
   StatusProcessAlarm : BOOL;   // UR20_16DO_P generic Module Data StatusProcessAlarm
END_STRUCT
END_TYPE

TYPE UDT_020_O :   // UR20_FBC_EIP Module UR20_FBC_EIP UDT for UR20_16DO_P Order No.: 1315250000 generic Module Data (Outputs)
STRUCT
   Data : UDT_020_Data_O;   // UR20_16DO_P generic Module Data Data
END_STRUCT
END_TYPE

TYPE UDT_045_Data_I :   // UR20_FBC_EIP Module UR20_FBC_EIP UDT for UR20_4AI_UI_16 Order No.: 1315620000 Process Data (Inputs)
STRUCT
   Ch_00 : INT;   // UR20_4AI_UI_16 Process Data Ch_00
   Ch_01 : INT;   // UR20_4AI_UI_16 Process Data Ch_01
   Ch_02 : INT;   // UR20_4AI_UI_16 Process Data Ch_02
   Ch_03 : INT;   // UR20_4AI_UI_16 Process Data Ch_03
END_STRUCT
END_TYPE

TYPE UDT_045_I :   // UR20_FBC_EIP Module UR20_FBC_EIP UDT for UR20_4AI_UI_16 Order No.: 1315620000 generic Module Data (Inputs)
STRUCT
   Data : UDT_045_Data_I;   // UR20_4AI_UI_16 generic Module Data Data
   Diagnostic : UDT_Diagnostic;   // UR20_4AI_UI_16 generic Module Data Diagnostic
   ProcessAlarm : UDT_ProcessAlarm;   // UR20_4AI_UI_16 generic Module Data ProcessAlarm
   StatusDiagAlarm : BOOL;   // UR20_4AI_UI_16 generic Module Data StatusDiagAlarm
   StatusProcessAlarm : BOOL;   // UR20_4AI_UI_16 generic Module Data StatusProcessAlarm
END_STRUCT
END_TYPE

TYPE UDT_045_O :   // UR20_FBC_EIP Module UR20_FBC_EIP UDT for UR20_4AI_UI_16 Order No.: 1315620000 generic Module Data (Outputs)
STRUCT
   Parameter : UDT_045_Parameter;   // UR20_4AI_UI_16 generic Module Data Parameter
END_STRUCT
END_TYPE

TYPE UDT_045_Parameter :   // UR20_FBC_EIP Module UR20_FBC_EIP UDT for UR20_4AI_UI_16 Order No.: 1315620000 Parameter Data (NOP)
STRUCT
   Frequency_suppression : INT;   // disabled-0x00 50 Hz-0x02 60 Hz-0x01 Average over 16 values-0x03 2 Hz low pass-0x04
   Ch_00_Data_format : BOOL;   // S5 data format-0x00 S7 data format-0x01
   Ch_00_Measurement_range : INT;   // 0 .. 20mA-0x85 4mA-20mA-0x87 0 .. 10V-0x01 -10 .. 10V-0x03 0V .. 5V-0x09 -5 .. 5V-0x0a 1V-5V-0x0b 2V-10V-0x02 Disabled-0xff
   Ch_01_Data_format : BOOL;   // S5 data format-0x00 S7 data format-0x01
   Ch_01_Measurement_range : INT;   // 0 .. 20mA-0x85 4mA-20mA-0x87 0 .. 10V-0x01 -10 .. 10V-0x03 0V .. 5V-0x09 -5 .. 5V-0x0a 1V-5V-0x0b 2V-10V-0x02 Disabled-0xff
   Ch_02_Data_format : BOOL;   // S5 data format-0x00 S7 data format-0x01
   Ch_02_Measurement_range : INT;   // 0 .. 20mA-0x85 4mA-20mA-0x87 0 .. 10V-0x01 -10 .. 10V-0x03 0V .. 5V-0x09 -5 .. 5V-0x0a 1V-5V-0x0b 2V-10V-0x02 Disabled-0xff
   Ch_03_Data_format : BOOL;   // S5 data format-0x00 S7 data format-0x01
   Ch_03_Measurement_range : INT;   // 0 .. 20mA-0x85 4mA-20mA-0x87 0 .. 10V-0x01 -10 .. 10V-0x03 0V .. 5V-0x09 -5 .. 5V-0x0a 1V-5V-0x0b 2V-10V-0x02 Disabled-0xff
END_STRUCT
END_TYPE

TYPE UDT_Diagnostic :   // Diagnostic data Type
STRUCT
   Err_A : SINT;   // Error indicator
   ModTyp : SINT;   // Module type
   Err_C : SINT;   // Error byte 2
   Err_D : SINT;   // Error byte 3
   ChTyp : SINT;   // Channel type
   NumBit : SINT;   // Number of diagnostic bit per channel
   NumCh : SINT;   // Number of similar channels per module
   ChErr_0 : SINT;   // Channel error
   ChErr_1 : SINT;   // Channel error
   ChErr_2 : SINT;   // Channel error
   ChErr_3 : SINT;   // Channel error
   Ch00Err : SINT;   // Error channel 00
   Ch01Err : SINT;   // Error channel 01
   Ch02Err : SINT;   // Error channel 02
   Ch03Err : SINT;   // Error channel 03
   Ch04Err : SINT;   // Error channel 04
   Ch05Err : SINT;   // Error channel 05
   Ch06Err : SINT;   // Error channel 06
   Ch07Err : SINT;   // Error channel 07
   Ch08Err : SINT;   // Error channel 08
   Ch09Err : SINT;   // Error channel 09
   Ch10Err : SINT;   // Error channel 10
   Ch11Err : SINT;   // Error channel 11
   Ch12Err : SINT;   // Error channel 12
   Ch13Err : SINT;   // Error channel 13
   Ch14Err : SINT;   // Error channel 14
   Ch15Err : SINT;   // Error channel 15
   Ch16Err : SINT;   // Error channel 16
   Ch17Err : SINT;   // Error channel 17
   Ch18Err : SINT;   // Error channel 18
   Ch19Err : SINT;   // Error channel 19
   Ch20Err : SINT;   // Error channel 20
   Ch21Err : SINT;   // Error channel 21
   Ch22Err : SINT;   // Error channel 22
   Ch23Err : SINT;   // Error channel 23
   Ch24Err : SINT;   // Error channel 24
   Ch25Err : SINT;   // Error channel 25
   Ch26Err : SINT;   // Error channel 26
   Ch27Err : SINT;   // Error channel 27
   Ch28Err : SINT;   // Error channel 28
   Ch29Err : SINT;   // Error channel 29
   Ch30Err : SINT;   // Error channel 30
   Ch31Err : SINT;   // Error channel 31
   Diag_US_1 : SINT;   // Timestamp 32Bit 24-31
   Diag_US_2 : SINT;   // Timestamp 32Bit 16-23
   Diag_US_3 : SINT;   // Timestamp 32Bit 8-15
   Diag_US_4 : SINT;   // Timestamp 32Bit 0-7
END_STRUCT
END_TYPE

TYPE UDT_ID0 :   // 1st Station UR20_FBC_EIP
STRUCT
   IN : UDT_ID0_I;   // IN Data
   OUT : UDT_ID0_O;   // OUT Data
   Status : UDT_ID0_Statusword;   // Statusword
   MISC : UDT_ID0_MISC;   // MISC
   WriteParameter : BOOL;   // Write all Parameter values for all UR20_FBC_EIP Modules
   ReadParameter : BOOL;   // Read all Parameter values for all UR20_FBC_EIP Modules
   EditParameter : BOOL;   // Allowed Edit all Parameter values for all UR20_FBC_EIP Modules
   SetDefaultParameter : BOOL;   // Reset all module parameters to their default value
END_STRUCT
END_TYPE

TYPE UDT_ID0_I :   // I- Module UDTs
STRUCT
   M01_UR20_16DI_P : UDT_015_I;   // UDT for UR20_16DI_P- Module
   M02_UR20_16DI_P : UDT_015_I;   // UDT for UR20_16DI_P- Module
   M03_UR20_4AI_UI_16 : UDT_045_I;   // UDT for UR20_4AI_UI_16- Module
   M04_UR20_16DO_P : UDT_020_I;   // UDT for UR20_16DO_P- Module
   M05_UR20_16DO_P : UDT_020_I;   // UDT for UR20_16DO_P- Module
END_STRUCT
END_TYPE

TYPE UDT_ID0_MISC :   // MISC
STRUCT
   Help_Value_DINT : DINT;   // Help Tag for Swop Command
   Help_Value_INT : INT;   // Help Tag for Swop Command
   Wrk_LINT : DINT[2];
   ParameterArray : SINT[1350];
   ParameterArray_RX_TX : SINT[1350];
   Startup_Flag : BOOL;   // Clr at startup and set aufter first use
   Tmr_ProcessAlarm : TIMER;   // Timer for Reading Process Alarmvalues
   Tmr_Diag : TIMER;   // Timer for Reading Diagnostic Alarmvalues
   Tmr_SetDefault : TIMER;   // Timer for reset Set Default Flag
   ProcessAlarm : SINT[8];   // Array for Process Alarm Data
   DiagnosticAlarm : SINT[8];   // Array for Diagnoses Alarm Data
   DiagnosticData : SINT[47];   // Storrage Array for Diagnose Data
   ProcessAlarmData : SINT[4];   // Storrage Array for Diagnose Data
   InputBytes : DINT;   // Number of total input bytes
   OutputBytes : DINT;   // Number of total output bytes
   ParameterBytes : DINT;   // Number of total Parameter bytes
END_STRUCT
END_TYPE

TYPE UDT_ID0_O :   // O- Module UDTs
STRUCT
   M03_UR20_4AI_UI_16 : UDT_045_O;   // UDT for UR20_4AI_UI_16- Module
   M04_UR20_16DO_P : UDT_020_O;   // UDT for UR20_16DO_P- Module
   M05_UR20_16DO_P : UDT_020_O;   // UDT for UR20_16DO_P- Module
END_STRUCT
END_TYPE

TYPE UDT_ID0_Statusword :   // packed input process data
STRUCT
   Summarized_module_diagnosis : BOOL;   // A diagnosis is available for at least one module with diagnostics functionality.
   Pending : BOOL;   // More than one electronic unit or module has been removed from the station.
   Errorbit_2 : BOOL;   // Reserved bit 2, currently not used
   Systembus_error : BOOL;   // Error on the system bus. Communication with the connected modules is disrupted.
   Unacknowledged_diagnosis_alarm : BOOL;   // Unacknowledged diagnosis alarm
   Unacknowledged_process_alarm : BOOL;   // Unacknowledged process alarm
   IOConfiguration_error : BOOL;   // Deviation in the configuration. The module list has changed. The list of configured modules (Configured Module Ident List class 0x65 (101), instance 0x01 (1), attribute 0x70 (112)) differs from the module list detected by the coupler (Detected Module Ident List class 0x65 (101), instance 0x01 (1), attribute 0x6F (111)).
   Master_configuration_error : BOOL;   // Master configuration error. The list of configured modules (Configured Module Ident List class 0x65 (101), instance 0x01, attribute 0x70 (112)) differs significantly from the module list detected by the coupler (Detected Module Ident List class 0x65 (101), instance 0x01 (1), attribute 0x6F (111)) ab. No process data can be exchanged with the modules.
   Errorbit_8 : BOOL;   // Reserved bit 8, currently not used
   Errorbit_9 : BOOL;   // Reserved bit 9, currently not used
   Force_mode_active : BOOL;   // Force mode was activated via web server. Process data cannot be exchanged between the master and forced channels
   Module_Pulled : BOOL;   // At least one module is pulled
   Errorbit_12 : BOOL;   // Reserved bit 12, currently not used
   Voltage_Uout_error : BOOL;   // Error in the voltage supply of output current path
   Voltage_Uin_error : BOOL;   // Error in the voltage supply of system and input current path
   Errorbit_15 : BOOL;   // Reserved bit 15, currently not used
END_STRUCT
END_TYPE

TYPE UDT_ID86 :   // 1st Station UR20_FBC_EIP
STRUCT
   IN : UDT_ID86_I;   // IN Data
   OUT : UDT_ID86_O;   // OUT Data
   Status : UDT_ID86_Statusword;   // Statusword
   MISC : UDT_ID86_MISC;   // MISC
   WriteParameter : BOOL;   // Write all Parameter values for all UR20_FBC_EIP Modules
   ReadParameter : BOOL;   // Read all Parameter values for all UR20_FBC_EIP Modules
   EditParameter : BOOL;   // Allowed Edit all Parameter values for all UR20_FBC_EIP Modules
   SetDefaultParameter : BOOL;   // Reset all module parameters to their default value
END_STRUCT
END_TYPE

TYPE UDT_ID86_I :   // I- Module UDTs
STRUCT
   M01_UR20_16DI_P : UDT_015_I;   // UDT for UR20_16DI_P- Module
   M02_UR20_16DI_P : UDT_015_I;   // UDT for UR20_16DI_P- Module
   M03_UR20_4AI_UI_16 : UDT_045_I;   // UDT for UR20_4AI_UI_16- Module
   M04_UR20_16DO_P : UDT_020_I;   // UDT for UR20_16DO_P- Module
   M05_UR20_16DO_P : UDT_020_I;   // UDT for UR20_16DO_P- Module
END_STRUCT
END_TYPE

TYPE UDT_ID86_MISC :   // MISC
STRUCT
   Help_Value_DINT : DINT;   // Help Tag for Swop Command
   Help_Value_INT : INT;   // Help Tag for Swop Command
   Wrk_LINT : DINT[2];
   ParameterArray : SINT[1350];
   ParameterArray_RX_TX : SINT[1350];
   Startup_Flag : BOOL;   // Clr at startup and set aufter first use
   Tmr_ProcessAlarm : TIMER;   // Timer for Reading Process Alarmvalues
   Tmr_Diag : TIMER;   // Timer for Reading Diagnostic Alarmvalues
   Tmr_SetDefault : TIMER;   // Timer for reset Set Default Flag
   ProcessAlarm : SINT[8];   // Array for Process Alarm Data
   DiagnosticAlarm : SINT[8];   // Array for Diagnoses Alarm Data
   DiagnosticData : SINT[47];   // Storrage Array for Diagnose Data
   ProcessAlarmData : SINT[4];   // Storrage Array for Diagnose Data
   InputBytes : DINT;   // Number of total input bytes
   OutputBytes : DINT;   // Number of total output bytes
   ParameterBytes : DINT;   // Number of total Parameter bytes
END_STRUCT
END_TYPE

TYPE UDT_ID86_O :   // O- Module UDTs
STRUCT
   M03_UR20_4AI_UI_16 : UDT_045_O;   // UDT for UR20_4AI_UI_16- Module
   M04_UR20_16DO_P : UDT_020_O;   // UDT for UR20_16DO_P- Module
   M05_UR20_16DO_P : UDT_020_O;   // UDT for UR20_16DO_P- Module
END_STRUCT
END_TYPE

TYPE UDT_ID86_Statusword :   // packed input process data
STRUCT
   Summarized_module_diagnosis : BOOL;   // A diagnosis is available for at least one module with diagnostics functionality.
   Pending : BOOL;   // More than one electronic unit or module has been removed from the station.
   Errorbit_2 : BOOL;   // Reserved bit 2, currently not used
   Systembus_error : BOOL;   // Error on the system bus. Communication with the connected modules is disrupted.
   Unacknowledged_diagnosis_alarm : BOOL;   // Unacknowledged diagnosis alarm
   Unacknowledged_process_alarm : BOOL;   // Unacknowledged process alarm
   IOConfiguration_error : BOOL;   // Deviation in the configuration. The module list has changed. The list of configured modules (Configured Module Ident List class 0x65 (101), instance 0x01 (1), attribute 0x70 (112)) differs from the module list detected by the coupler (Detected Module Ident List class 0x65 (101), instance 0x01 (1), attribute 0x6F (111)).
   Master_configuration_error : BOOL;   // Master configuration error. The list of configured modules (Configured Module Ident List class 0x65 (101), instance 0x01, attribute 0x70 (112)) differs significantly from the module list detected by the coupler (Detected Module Ident List class 0x65 (101), instance 0x01 (1), attribute 0x6F (111)) ab. No process data can be exchanged with the modules.
   Errorbit_8 : BOOL;   // Reserved bit 8, currently not used
   Errorbit_9 : BOOL;   // Reserved bit 9, currently not used
   Force_mode_active : BOOL;   // Force mode was activated via web server. Process data cannot be exchanged between the master and forced channels
   Module_Pulled : BOOL;   // At least one module is pulled
   Errorbit_12 : BOOL;   // Reserved bit 12, currently not used
   Voltage_Uout_error : BOOL;   // Error in the voltage supply of output current path
   Voltage_Uin_error : BOOL;   // Error in the voltage supply of system and input current path
   Errorbit_15 : BOOL;   // Reserved bit 15, currently not used
END_STRUCT
END_TYPE

TYPE UDT_ProcessAlarm :   // ProcessAlarm data Type
STRUCT
   PRIT_OL : SINT;
   PRIT_UL : SINT;
   PRIT_US0 : SINT;
   PRIT_US1 : SINT;
END_STRUCT
END_TYPE

TYPE VFD :
STRUCT
   Ramp : REAL;
   Speed : INT;
   Run : BOOL;
   Running : BOOL;
   Ready : BOOL;
   Stop : BOOL;
   Current_speed : INT;
END_STRUCT
END_TYPE

TYPE Vision :
STRUCT
   Enable : BOOL;
   Trigger : BOOL;
   Result_OK : BOOL;
   Result_NG : BOOL;
   Ready : BOOL;
   Result_Ready : BOOL;
   Busy : BOOL;
   Prog : SINT;
   Current_Prog : SINT;
   Trigger_ON_TM : TIMER;
   Trigger_OFF_TM : TIMER;
END_STRUCT
END_TYPE

ADD_ON_INSTRUCTION AlicatCommand   (* revision 1.0, vendor Alicat Scientific, Inc *)
// Executes a command through CIP explicit messaging.
// Help:
// Executes an Alicat asynchronous command by sending CIP explicit message commands to the device.
// Reqires a Controller tag of type INT[2] to store data written to/read from the device.
// Requires two MESSAGE tags configured in the following way:
// RequestMsg:
//   CIP Generic - Get Attribute Single
//   Class 4, Instance 102, Attribute 3
//   Source: CmdData
//   Length: 4
// Response Msg:
//   CIP Generic: Get Attribute Single
//   Class 4, Instance 103, Attribute 3
//   Destination: CmdData
// The command is triggered on transition of the START bit from 0 to 1. CmdID and CmdArg are passed to the device. Upon completion, EnableOut is set and the command result is copied into CmdResult. If an error occurs in one of the explicit messages the ER bit will be set.
// Setting the START bit before EnableOut is set from the previous command will have unpredictable effects.
VAR_IN_OUT
   RequestMsg : MESSAGE; {required}
   ResponseMsg : MESSAGE; {required}
   CmdData : INT[2]; {required}
END_VAR
VAR_INPUT
   CmdID : INT; {visible}
   CmdArg : INT; {visible}
END_VAR
VAR_OUTPUT
   CmdResult : INT; {access Read Only, visible}
   ER : BOOL; {access Read Only, visible}
END_VAR
VAR_INPUT
   START : ALIAS FOR CmdTrigger.0; {access None}
END_VAR
VAR
   CmdTrigger : DINT; {access None}
END_VAR

ROUTINE Logic   (* ladder *)
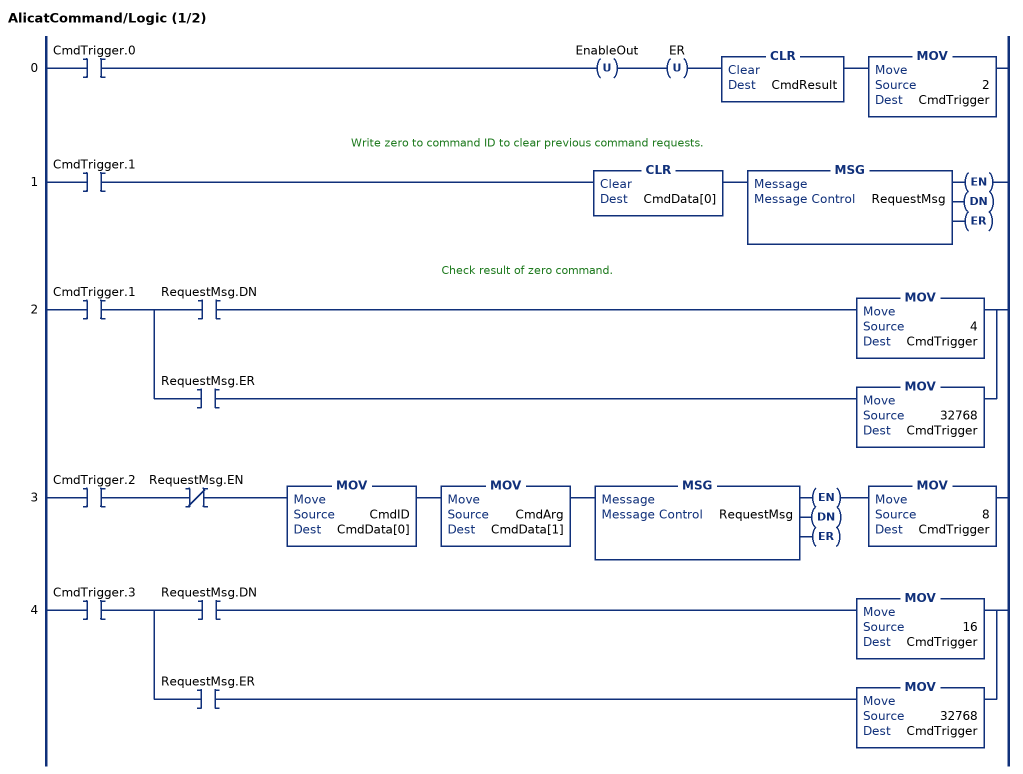
   0: XIC(CmdTrigger.0)OTU(EnableOut)OTU(ER)CLR(CmdResult)MOV(2,CmdTrigger);
   // Write zero to command ID to clear previous command requests.
   1: XIC(CmdTrigger.1)CLR(CmdData[0])MSG(RequestMsg);
   // Check result of zero command.
   2: XIC(CmdTrigger.1)[XIC(RequestMsg.DN) MOV(4,CmdTrigger) ,XIC(RequestMsg.ER) MOV(32768,CmdTrigger) ];
   3: XIC(CmdTrigger.2)XIO(RequestMsg.EN)MOV(CmdID,CmdData[0])MOV(CmdArg,CmdData[1])MSG(RequestMsg)MOV(8,CmdTrigger);
   4: XIC(CmdTrigger.3)[XIC(RequestMsg.DN) MOV(16,CmdTrigger) ,XIC(RequestMsg.ER) MOV(32768,CmdTrigger) ];
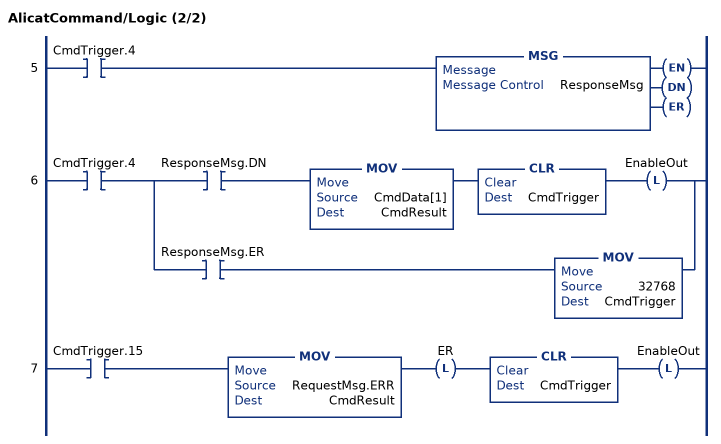
   5: XIC(CmdTrigger.4)MSG(ResponseMsg);
   6: XIC(CmdTrigger.4)[XIC(ResponseMsg.DN) MOV(CmdData[1],CmdResult) CLR(CmdTrigger) OTL(EnableOut) ,XIC(ResponseMsg.ER) MOV(32768,CmdTrigger) ];
   7: XIC(CmdTrigger.15)MOV(RequestMsg.ERR,CmdResult)OTL(ER)CLR(CmdTrigger)OTL(EnableOut);
END_ROUTINE
END_ADD_ON_INSTRUCTION

ADD_ON_INSTRUCTION AlicatUpdateInput   (* revision 1.0, vendor Alicat Scientific, Inc *)
// Updates AlicatIoData UDT from device input data array.
// Help:
// This AOI copies input data from an Alicat IO device into a UDT which allows accessing data readings as REAL values. It also decodes the device status word into status flags. Since RSLogix performs device IO asynchronously, it is recommended to copy the input data into a SINT array with the CPS instruction before calling this AOI.
// Before calling, set the flags in IoData.Config to match the configuration of your device. See the Alicat operating bulletin for more information.
VAR_IN_OUT
   InputArray : SINT[6]; {required}   // Array of SINTs from device input data.
   IoData : AlicatIoData; {required}   // AlicatIoData UDT to update.
END_VAR
VAR
   InputSize : DINT; {access None}
   InputOffset : DINT; {access None}
END_VAR

ROUTINE Logic   (* ladder *)
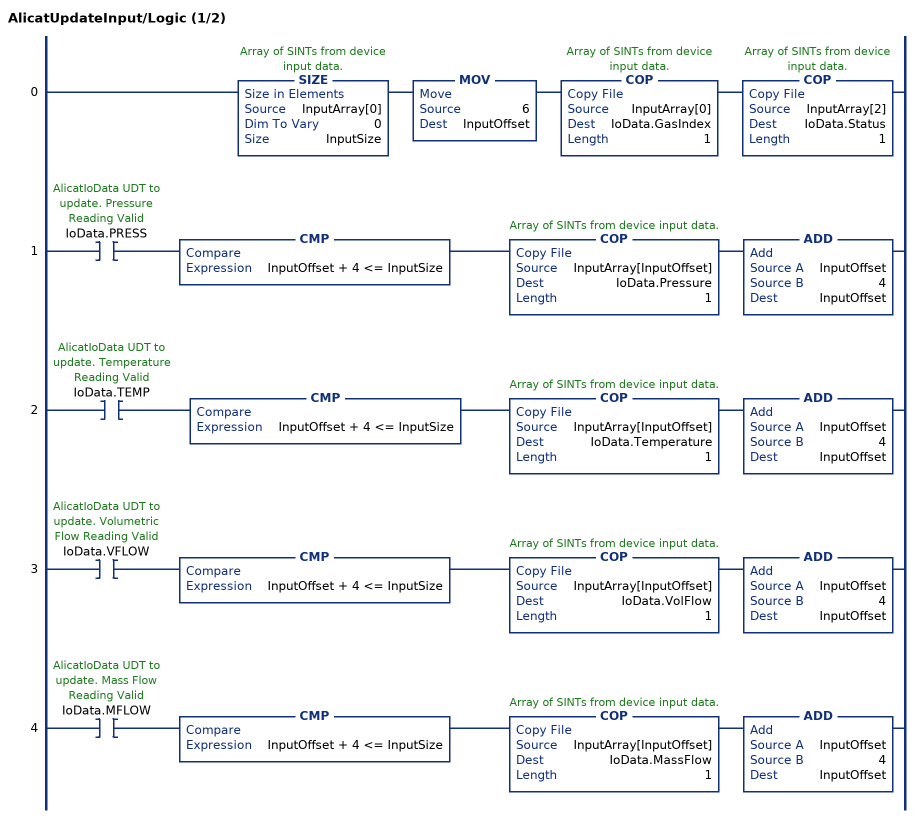
   0: SIZE(InputArray[0],0,InputSize)MOV(6,InputOffset)COP(InputArray[0],IoData.GasIndex,1)COP(InputArray[2],IoData.Status,1);
   1: XIC(IoData.PRESS)CMP(InputOffset + 4 <= InputSize)COP(InputArray[InputOffset],IoData.Pressure,1)ADD(InputOffset,4,InputOffset);
   2: XIC(IoData.TEMP)CMP(InputOffset + 4 <= InputSize)COP(InputArray[InputOffset],IoData.Temperature,1)ADD(InputOffset,4,InputOffset);
   3: XIC(IoData.VFLOW)CMP(InputOffset + 4 <= InputSize)COP(InputArray[InputOffset],IoData.VolFlow,1)ADD(InputOffset,4,InputOffset);
   4: XIC(IoData.MFLOW)CMP(InputOffset + 4 <= InputSize)COP(InputArray[InputOffset],IoData.MassFlow,1)ADD(InputOffset,4,InputOffset);
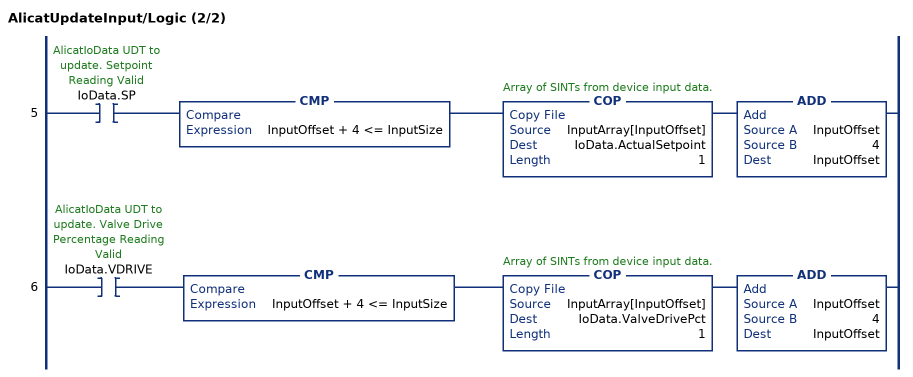
   5: XIC(IoData.SP)CMP(InputOffset + 4 <= InputSize)COP(InputArray[InputOffset],IoData.ActualSetpoint,1)ADD(InputOffset,4,InputOffset);
   6: XIC(IoData.VDRIVE)CMP(InputOffset + 4 <= InputSize)COP(InputArray[InputOffset],IoData.ValveDrivePct,1)ADD(InputOffset,4,InputOffset);
END_ROUTINE
END_ADD_ON_INSTRUCTION

ADD_ON_INSTRUCTION AOI_DIG_INPUT_DEB   (* revision 1.0, ExecuteEnableInFalse *)
VAR_INPUT
   INPUT : BOOL; {required}
   RESET : BOOL; {required}
   ON_TIME : REAL; {required}
   OFF_TIME : REAL; {required}
END_VAR
VAR_OUTPUT
   DEB_INPUT : BOOL; {access Read Only, visible}
   IN : BOOL; {access Read Only}
   ON_TT : BOOL; {access Read Only}
   OFF_TT : BOOL; {access Read Only}
   OUT : BOOL; {access Read Only}
END_VAR
VAR
   OFF_TMR : TIMER; {access None}
   ON_TMR : TIMER; {access None}
   RESET_ONS : BOOL; {access None}
END_VAR

ROUTINE EnableInFalse   (* ladder *)
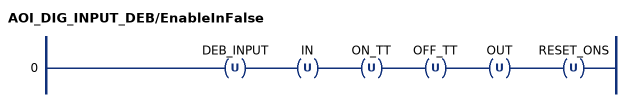
   0: OTU(DEB_INPUT)OTU(IN)OTU(ON_TT)OTU(OFF_TT)OTU(OUT)OTU(RESET_ONS);
END_ROUTINE

ROUTINE Logic   (* ladder *)
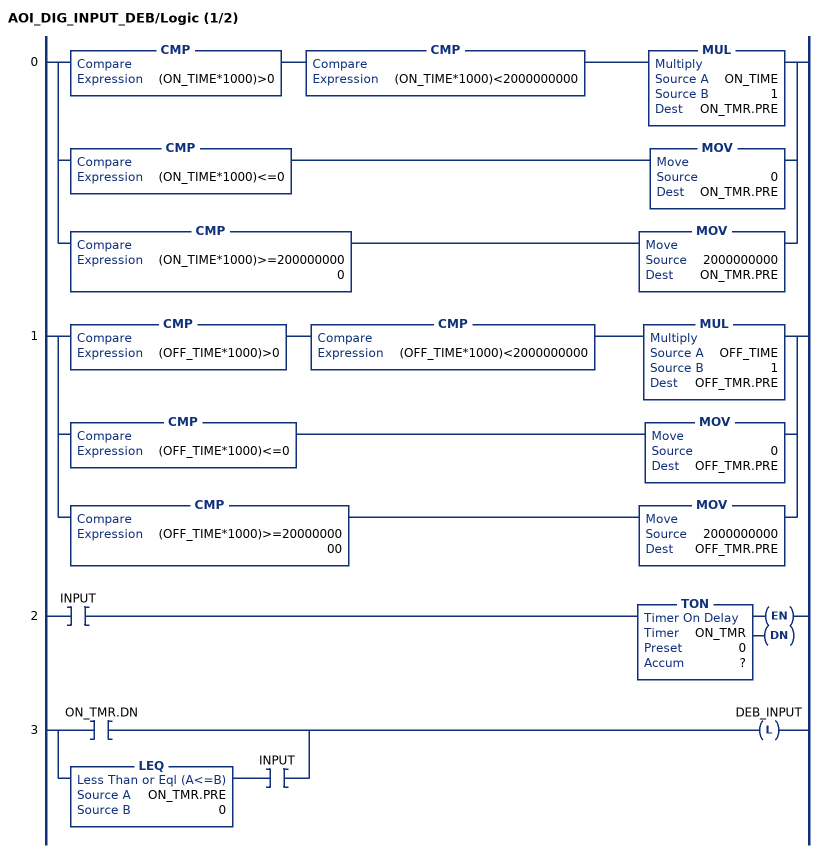
   0: [CMP((ON_TIME*1000)>0) CMP((ON_TIME*1000)<2000000000) MUL(ON_TIME,1,ON_TMR.PRE) ,CMP((ON_TIME*1000)<=0) MOV(0,ON_TMR.PRE) ,CMP((ON_TIME*1000)>=2000000000) MOV(2000000000,ON_TMR.PRE) ];
   1: [CMP((OFF_TIME*1000)>0) CMP((OFF_TIME*1000)<2000000000) MUL(OFF_TIME,1,OFF_TMR.PRE) ,CMP((OFF_TIME*1000)<=0) MOV(0,OFF_TMR.PRE) ,CMP((OFF_TIME*1000)>=2000000000) MOV(2000000000,OFF_TMR.PRE) ];
   2: XIC(INPUT)TON(ON_TMR,?,?);
   3: [XIC(ON_TMR.DN) ,LEQ(ON_TMR.PRE,0) XIC(INPUT) ]OTL(DEB_INPUT);
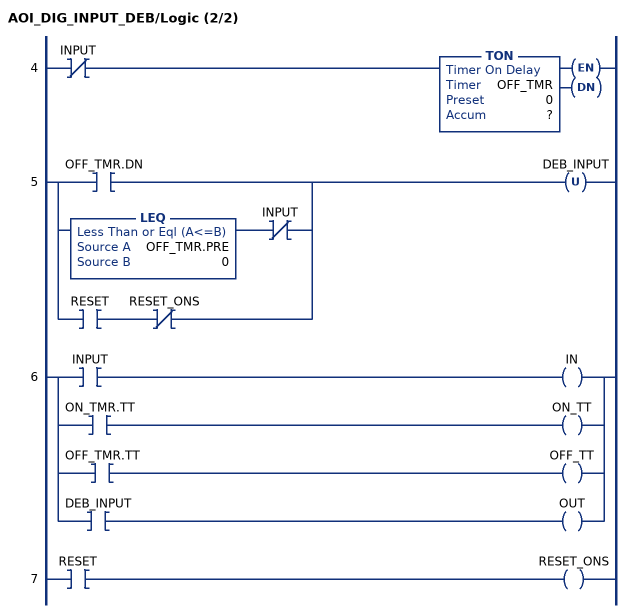
   4: XIO(INPUT)TON(OFF_TMR,?,?);
   5: [XIC(OFF_TMR.DN) ,LEQ(OFF_TMR.PRE,0) XIO(INPUT) ,XIC(RESET) XIO(RESET_ONS) ]OTU(DEB_INPUT);
   6: [XIC(INPUT) OTE(IN) ,XIC(ON_TMR.TT) OTE(ON_TT) ,XIC(OFF_TMR.TT) OTE(OFF_TT) ,XIC(DEB_INPUT) OTE(OUT) ];
   7: XIC(RESET)OTE(RESET_ONS);
END_ROUTINE
END_ADD_ON_INSTRUCTION

ADD_ON_INSTRUCTION Banner_XS26_Fault_Log_Read   (* revision 1.0, vendor Banner Engineering *)
// This AOI uses Explicit Messaging to read the Fault Log of a XS26 or SC26 controller.
VAR_IN_OUT
   Routine_Bit_Control : BOOL; {required}
   Fault_Log_1 : MESSAGE; {required}
   Fault_Log_2 : MESSAGE; {required}
   Fault_Log_3 : MESSAGE; {required}
   Fault_Log_4 : MESSAGE; {required}
   Fault_Log_5 : MESSAGE; {required}
   Fault_Log_6 : MESSAGE; {required}
   Fault_Log_7 : MESSAGE; {required}
   Fault_Log_8 : MESSAGE; {required}
   Fault_Log_9 : MESSAGE; {required}
   Fault_Log_10 : MESSAGE; {required}
END_VAR
VAR
   Lock_Flag : DINT; {access None}
END_VAR

ROUTINE Logic   (* ladder *)
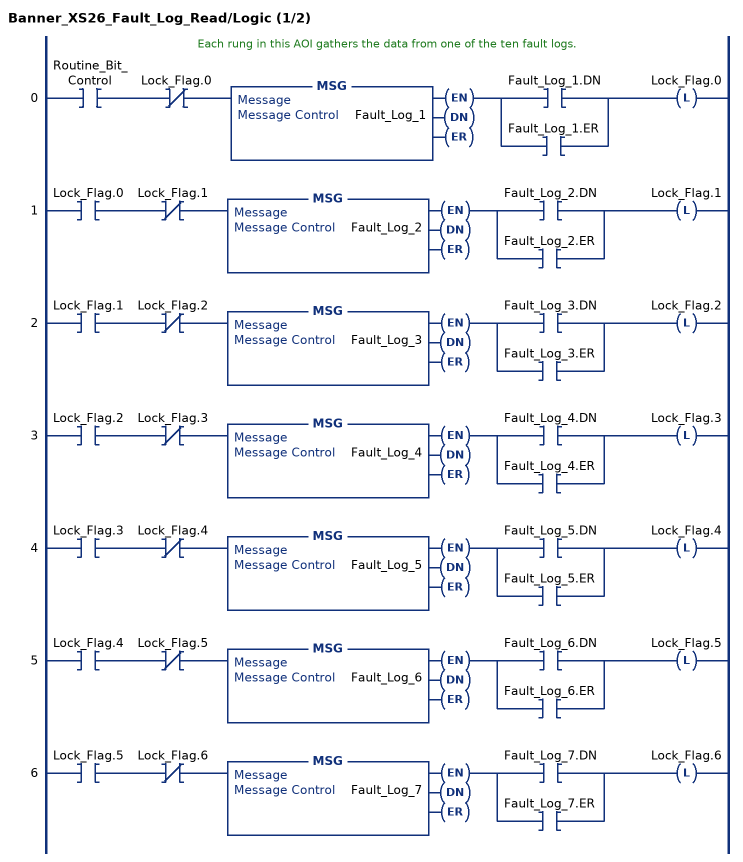
   // Each rung in this AOI gathers the data from one of the ten fault logs.
   0: XIC(Routine_Bit_Control)XIO(Lock_Flag.0)MSG(Fault_Log_1)[XIC(Fault_Log_1.DN) ,XIC(Fault_Log_1.ER) ]OTL(Lock_Flag.0);
   1: XIC(Lock_Flag.0)XIO(Lock_Flag.1)MSG(Fault_Log_2)[XIC(Fault_Log_2.DN) ,XIC(Fault_Log_2.ER) ]OTL(Lock_Flag.1);
   2: XIC(Lock_Flag.1)XIO(Lock_Flag.2)MSG(Fault_Log_3)[XIC(Fault_Log_3.DN) ,XIC(Fault_Log_3.ER) ]OTL(Lock_Flag.2);
   3: XIC(Lock_Flag.2)XIO(Lock_Flag.3)MSG(Fault_Log_4)[XIC(Fault_Log_4.DN) ,XIC(Fault_Log_4.ER) ]OTL(Lock_Flag.3);
   4: XIC(Lock_Flag.3)XIO(Lock_Flag.4)MSG(Fault_Log_5)[XIC(Fault_Log_5.DN) ,XIC(Fault_Log_5.ER) ]OTL(Lock_Flag.4);
   5: XIC(Lock_Flag.4)XIO(Lock_Flag.5)MSG(Fault_Log_6)[XIC(Fault_Log_6.DN) ,XIC(Fault_Log_6.ER) ]OTL(Lock_Flag.5);
   6: XIC(Lock_Flag.5)XIO(Lock_Flag.6)MSG(Fault_Log_7)[XIC(Fault_Log_7.DN) ,XIC(Fault_Log_7.ER) ]OTL(Lock_Flag.6);
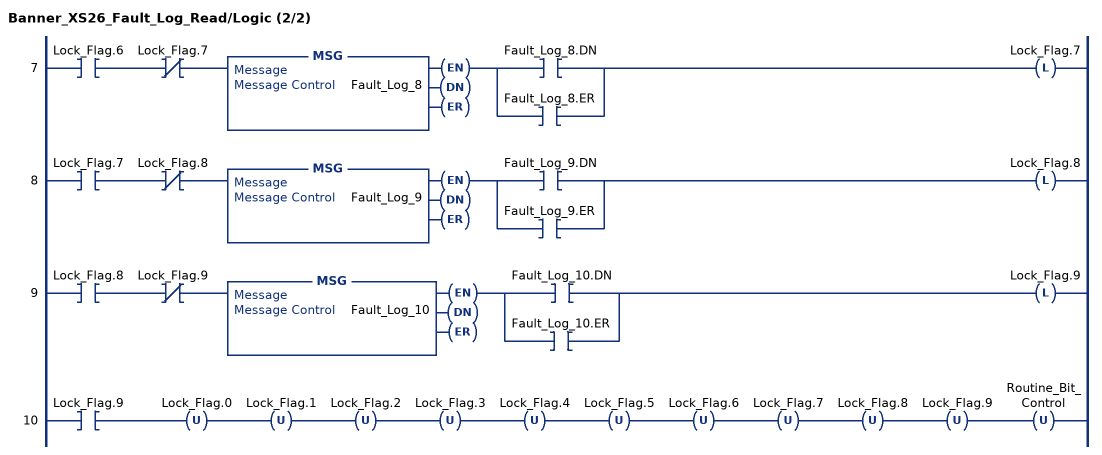
   7: XIC(Lock_Flag.6)XIO(Lock_Flag.7)MSG(Fault_Log_8)[XIC(Fault_Log_8.DN) ,XIC(Fault_Log_8.ER) ]OTL(Lock_Flag.7);
   8: XIC(Lock_Flag.7)XIO(Lock_Flag.8)MSG(Fault_Log_9)[XIC(Fault_Log_9.DN) ,XIC(Fault_Log_9.ER) ]OTL(Lock_Flag.8);
   9: XIC(Lock_Flag.8)XIO(Lock_Flag.9)MSG(Fault_Log_10)[XIC(Fault_Log_10.DN) ,XIC(Fault_Log_10.ER) ]OTL(Lock_Flag.9);
   10: XIC(Lock_Flag.9)OTU(Lock_Flag.0)OTU(Lock_Flag.1)OTU(Lock_Flag.2)OTU(Lock_Flag.3)OTU(Lock_Flag.4)OTU(Lock_Flag.5)OTU(Lock_Flag.6)OTU(Lock_Flag.7)OTU(Lock_Flag.8)OTU(Lock_Flag.9)OTU(Routine_Bit_Control);
END_ROUTINE
END_ADD_ON_INSTRUCTION
